// TIA Portal V19 export
TYPE "LEXCHANGETRAY_typeConstraintRollerEm_toHandlingXyzDeliver"
// stored: Access Published
   STRUCT
      feedback : "LEXCHANGETRAY_typeConstraintRollerEm_toHandlingXyzFeedback";
      req : "LEXCHANGETRAY_typeConstraintRollerEm_toHandlingXyzReq";
   END_STRUCT;
END_TYPE
